{attribute 'Tc2GvlVarNames'}
VAR_GLOBAL RETAIN

END_VAR

(* stored: Version 1.1.0.1, ProductVersion 3.1.4022.7
   GVL Setup_Data: Id {00a0fbaa-2260-496e-aeb1-b0524c2f3478} *)
